FUNCTION TryConvert_INT_TO_LINT : BOOL
VAR_INPUT
	in : INT;
	out : REFERENCE TO LINT;
END_VAR

out := INT_TO_LINT(in);
TryConvert_INT_TO_LINT := TRUE;

END_FUNCTION

(* stored: Version 1.1.0.1, ProductVersion 3.1.4024.12
   POU TryConvert_INT_TO_LINT: Id {93d9abf0-d80b-4659-a39a-ae33c7466bff}, SpecialFunc None *)
